// TIA Portal V21 export
DATA_BLOCK "PidTemp_RiscaldamentoProdotto"   // DB43
// stored: InstanceOfName PID_Temp, OfSystemLibElement PID_Temp, OfSystemLibVersion 1.1
PID_Temp   // technology object, version 1.1
   // VAR_INPUT
   //    Setpoint : Real;
   //    Input : Real;
   //    Input_PER : Int;
   //    Disturbance : Real;
   //    ManualEnable : Bool;
   //    ManualValue : Real;
   //    ErrorAck : Bool;
   //    Reset : Bool;
   //    ModeActivate : Bool;
   // END_VAR
   // VAR_OUTPUT
   //    ScaledInput { ExternalWritable := 'False'} : Real;
   //    OutputHeat { ExternalWritable := 'False'} : Real;
   //    OutputCool { ExternalWritable := 'False'} : Real;
   //    OutputHeat_PER { ExternalWritable := 'False'} : Int;
   //    OutputCool_PER { ExternalWritable := 'False'} : Int;
   //    OutputHeat_PWM { ExternalWritable := 'False'} : Bool;
   //    OutputCool_PWM { ExternalWritable := 'False'} : Bool;
   //    SetpointLimit_H { ExternalWritable := 'False'} : Bool;
   //    SetpointLimit_L { ExternalWritable := 'False'} : Bool;
   //    InputWarning_H { ExternalWritable := 'False'} : Bool;
   //    InputWarning_L { ExternalWritable := 'False'} : Bool;
   //    State { ExternalWritable := 'False'} : Int;
   //    Error { ExternalWritable := 'False'} : Bool;
   //    ErrorBits { ExternalWritable := 'False'} : DWord;
   // END_VAR
   // VAR_IN_OUT
   //    Mode : Int := 3;
   //    Master : DWord;
   //    Slave : DWord;
   // END_VAR
   // VAR
   //    InternalDiagnostic : DWord;
   //    InternalVersion { ExternalWritable := 'False'} : DWord;
   //    InternalRTVersion : DWord;
   //    IntegralResetMode { S7_SetPoint := 'True'} : Int;
   //    OverwriteInitialOutputValue : Real;
   //    RunModeByStartup { S7_SetPoint := 'True'} : Bool;
   //    LoadBackUp : Bool;
   //    SetSubstituteOutput { S7_SetPoint := 'True'} : Bool;
   //    PhysicalUnit { ExternalWritable := 'False'; S7_SetPoint := 'True'} : Int;
   //    PhysicalQuantity { ExternalWritable := 'False'; S7_SetPoint := 'True'} : Int;
   //    ActivateRecoverMode { S7_SetPoint := 'True'} : Bool;
   // END_VAR
   // VAR RETAIN
   //    Warning { ExternalWritable := 'False'} : DWord;
   //    WarningInternal { ExternalWritable := 'False'} : DWord;
   // END_VAR
   // VAR
   //    Progress { ExternalWritable := 'False'} : Real;
   //    CurrentSetpoint { ExternalWritable := 'False'} : Real;
   //    CancelTuningLevel { S7_SetPoint := 'True'} : Real;
   //    SubstituteOutput { S7_SetPoint := 'True'} : Real;
   //    PidOutputSum { ExternalWritable := 'False'} : Real;
   //    PidOutputOffsetHeat { S7_SetPoint := 'True'} : Real;
   //    PidOutputOffsetCool { S7_SetPoint := 'True'} : Real;
   //    SubstituteSetpointOn { S7_SetPoint := 'True'} : Bool;
   //    SubstituteSetpoint { S7_SetPoint := 'True'} : Real;
   //    DisableCooling { S7_SetPoint := 'True'} : Bool;
   //    AllSlaveAutomaticState { ExternalWritable := 'False'} : Bool;
   //    NoSlaveSubstituteSetpoint { ExternalWritable := 'False'} : Bool;
   //    Heat { S7_SetPoint := 'True'} : PID_TempBasicOutputData;
   //    Cool { S7_SetPoint := 'True'} : PID_TempBasicOutputData;
   //    Config { S7_SetPoint := 'True'} : PID_TempConfig;
   //    CycleTime { S7_SetPoint := 'True'} : PID_CycleTime;
   //    CtrlParamsBackUp { S7_SetPoint := 'True'} : PID_TempControlParamsHeatCool;
   //    PIDSelfTune { S7_SetPoint := 'True'} : PID_TempSelfTune;
   //    PIDCtrl { S7_SetPoint := 'True'} : PID_TempControl;
   // END_VAR
   // VAR RETAIN
   //    Retain { S7_SetPoint := 'True'} : PID_TempRetain;
   // END_VAR
BEGIN
   Config.InputPerOn := FALSE;
   Config.Output.Heat.Select := 0;
   Config.Cascade.IsMaster := TRUE;
END_DATA_BLOCK
